VAR_GLOBAL
	g_IOCHostIP	: T_IPv4Addr := "127.0.0.1";
	g_udpMessengerPort	:	UDINT := 5555;
END_VAR

(* stored: Version 1.1.0.1, ProductVersion 3.1.4018.5
   GVL GVL_Messenger: Id {047a20cc-a785-4614-8465-ede098785b35} *)
